(* IEC 61131-3 sources: taveren/tests/fixtures/water_tank_sfc_one_sensor/build, 2 files *)

(* ---- plc.st ---- *)
TYPE
  LOGLEVEL : (CRITICAL, WARNING, INFO, DEBUG) := INFO;
END_TYPE

FUNCTION_BLOCK LOGGER
  VAR_INPUT
    TRIG : BOOL;
    MSG : STRING;
    LEVEL : LOGLEVEL := INFO;
  END_VAR
  VAR
    TRIG0 : BOOL;
  END_VAR

  IF TRIG AND NOT TRIG0 THEN
  {{
   LogMessage(GetFbVar(LEVEL),(char*)GetFbVar(MSG, .body),GetFbVar(MSG, .len));
  }}
  END_IF;
  TRIG0:=TRIG;
END_FUNCTION_BLOCK

FUNCTION_BLOCK python_eval
  VAR_INPUT
    TRIG : BOOL;
    CODE : STRING;
  END_VAR
  VAR_OUTPUT
    ACK : BOOL;
    RESULT : STRING;
  END_VAR
  VAR
    STATE : DWORD;
    BUFFER : STRING;
    PREBUFFER : STRING;
    TRIGM1 : BOOL;
    TRIGGED : BOOL;
  END_VAR

  {extern void __PythonEvalFB(int, PYTHON_EVAL*);__PythonEvalFB(0, data__);}
END_FUNCTION_BLOCK

FUNCTION_BLOCK python_poll
  VAR_INPUT
    TRIG : BOOL;
    CODE : STRING;
  END_VAR
  VAR_OUTPUT
    ACK : BOOL;
    RESULT : STRING;
  END_VAR
  VAR
    STATE : DWORD;
    BUFFER : STRING;
    PREBUFFER : STRING;
    TRIGM1 : BOOL;
    TRIGGED : BOOL;
  END_VAR

  {extern void __PythonEvalFB(int, PYTHON_EVAL*);__PythonEvalFB(1,(PYTHON_EVAL*)(void*)data__);}
END_FUNCTION_BLOCK

FUNCTION_BLOCK python_gear
  VAR_INPUT
    N : UINT;
    TRIG : BOOL;
    CODE : STRING;
  END_VAR
  VAR_OUTPUT
    ACK : BOOL;
    RESULT : STRING;
  END_VAR
  VAR
    py_eval : python_eval;
    COUNTER : UINT;
    _TMP_ADD10_OUT : UINT;
    _TMP_EQ13_OUT : BOOL;
    _TMP_SEL15_OUT : UINT;
    _TMP_AND7_OUT : BOOL;
  END_VAR

  _TMP_ADD10_OUT := ADD(COUNTER, 1);
  _TMP_EQ13_OUT := EQ(N, _TMP_ADD10_OUT);
  _TMP_SEL15_OUT := SEL(_TMP_EQ13_OUT, _TMP_ADD10_OUT, 0);
  COUNTER := _TMP_SEL15_OUT;
  _TMP_AND7_OUT := AND(_TMP_EQ13_OUT, TRIG);
  py_eval(TRIG := _TMP_AND7_OUT, CODE := CODE);
  ACK := py_eval.ACK;
  RESULT := py_eval.RESULT;
END_FUNCTION_BLOCK

TYPE
  datatype0 : BOOL;
END_TYPE

PROGRAM water_tank_sfc
  VAR
    low_level_sensor : SINT := 15;
    high_level_sensor : SINT := 85;
    motor : BOOL := False;
    water_level : SINT := 50;
  END_VAR

  INITIAL_STEP Initialize:
    motor(R);
  END_STEP

  TRANSITION FROM Initialize TO Fill_Tank
    := water_level < 15;
  END_TRANSITION

  STEP Fill_Tank:
    motor(N);
  END_STEP

  TRANSITION FROM Fill_Tank TO Stop_Motor
    := water_level > 85;
  END_TRANSITION

  STEP Stop_Motor:
    motor(R);
  END_STEP

  TRANSITION FROM Stop_Motor TO Fill_Tank
    := water_level < 15;
  END_TRANSITION

END_PROGRAM

CONFIGURATION Config0

  RESOURCE Res0 ON PLC
    TASK task0(INTERVAL := T#20ms,PRIORITY := 0);
    PROGRAM instance0 WITH task0 : water_tank_sfc;
  END_RESOURCE
END_CONFIGURATION

(* ---- generated_plc.st ---- *)
TYPE
  datatype0 : BOOL;
END_TYPE

PROGRAM water_tank_sfc
  VAR
    low_level_sensor : SINT := 15;
    high_level_sensor : SINT := 85;
    motor : BOOL := False;
    water_level : SINT := 50;
  END_VAR

  INITIAL_STEP Initialize:
    motor(R);
  END_STEP

  TRANSITION FROM Initialize TO Fill_Tank
    := water_level < 15;
  END_TRANSITION

  STEP Fill_Tank:
    motor(N);
  END_STEP

  TRANSITION FROM Fill_Tank TO Stop_Motor
    := water_level > 85;
  END_TRANSITION

  STEP Stop_Motor:
    motor(R);
  END_STEP

  TRANSITION FROM Stop_Motor TO Fill_Tank
    := water_level < 15;
  END_TRANSITION

END_PROGRAM

CONFIGURATION Config0

  RESOURCE Res0 ON PLC
    TASK task0(INTERVAL := T#20ms,PRIORITY := 0);
    PROGRAM instance0 WITH task0 : water_tank_sfc;
  END_RESOURCE
END_CONFIGURATION
